TYPE State :
STRUCT
	x : LREAL;
	y : LREAL;
	theta: LREAL;
END_STRUCT
END_TYPE

(* stored: Version 1.1.0.1, ProductVersion 3.1.4026.13
   DUT State: Id {7ee9265d-497c-40ce-b584-25f04dc4f39e} *)
